ABB RAPID module: BE_User.sys

%%%
  VERSION:1
  LANGUAGE:ENGLISH
%%%

MODULE BE_User(SYSMODULE)
    !
    ! 2007-07-01 S?
    !   CHG: Added data for tcp check freq. from BE_Mnu.
    ! 2006-01-17 S?
    !   CHG: Added data scanMig and tdMig for use in setup.
    !   CHG: Renamed procedures due to name conflicts with bullseye.
    ! 2006-01-13 S?
    !   CHG: Changed name to BE_User due to restore problem with BullsEye, name conflict
    !
    TASK PERS tooldata tWeldGun:=[TRUE,[[0,0,0],[1,0,0,0]],[1,[1,0,0],[1,0,0,0],0,0,0]];
    !
    LOCAL CONST jointtarget jtEmpty:=[[9E+09,9E+09,9E+09,9E+09,9E+09,9E+09],[9E+09,9E+09,9E+09,9E+09,9E+09,9E+09]];
    TASK PERS jointtarget jtBEHome:=[[94.4267,-36.8911,24.1644,-0.0315949,63.4412,0.285663],[4816.37,9E+09,9E+09,9E+09,9E+09,9E+09]];
    TASK PERS jointtarget jtBEApprPos:=[[144.389,0.963088,5.42986,-3.28422,43.5331,5.14622],[4816.37,9E+09,9E+09,9E+09,9E+09,9E+09]];
    TASK PERS jointtarget jtBEStartPos:=[[143.497,1.4308,11.9387,-2.84858,36.5204,4.36587],[4816.37,9E+09,9E+09,9E+09,9E+09,9E+09]];
    !
    !CONST be_device devUp:=["sen1",TRUE,[6,45,100,100],[40,45,100,100],0.10,FALSE,TRUE,TRUE];
    CONST be_device devUp:=["sen1",TRUE,[6,45,100,100],[40,45,100,100],0.10,FALSE,TRUE,TRUE];
    CONST be_device devDown:=["sen1",TRUE,[6,45,100,100],[40,45,100,100],0.10,TRUE,TRUE,TRUE];
    CONST be_scan scanMig:=[2,8,8,45,35,25];
    !CONST be_tooldesign tdMig:=[TRUE,30,18,50,6,6,TRUE,TRUE,1.2,[150,120,100,100],[250,150,100,100]];
    CONST be_tooldesign tdMig:=[TRUE,30,18,40,6,6,TRUE,TRUE,1.2,[150,120,100,100],[250,150,100,100]];
    !
    TASK PERS num nTcpExtension:=20;
    ! vars for tcp check during production
    TASK PERS num nBECheckTcpFreq:=0;
    TASK PERS num nBECheckCycle:=0;
    TASK PERS num numElapsedTime:=607.948;
    TASK PERS num numMeanDev:=0.0669059;
    TASK PERS num numMaxDev:=0.0974435;

    !
    PROC BEToolSetup()
        VAR jointtarget jCurrPos;
        VAR string sHeader;
        VAR string sMsg{5};
        VAR btnres nAnswer;

        sHeader:="BullsEye"+" ("+GetTaskName()+")";
        MoveAbsJ [[94.4267,-36.8911,24.1644,-0.0315949,63.4412,0.285663],[4816.37,9E+09,9E+09,9E+09,9E+09,9E+09]]\NoEOffs, v1000, z50, toolWeldGun1;
        sMsg{1}:="Press Yes to run setup for BullsEye scanning process.";
        sMsg{2}:="";
        sMsg{3}:="Press No to cancel.";
        sMsg{4}:="";
        sMsg{5}:="";
        UIMsgBox\Header:=sHeader,sMsg{1}\MsgLine2:=sMsg{2}\MsgLine3:=sMsg{3}\MsgLine4:=sMsg{4}\MsgLine5:=sMsg{5}\Buttons:=btnYesNo\Icon:=iconInfo\Result:=nAnswer;
        IF (nAnswer=resYes) THEN
            !The length of the TCP extension, as measured from the end of the tool body, is defined
            !here in millimeters.
            sHeader:="BullsEye"+" ("+GetTaskName()+")";
            sMsg{1}:="TCP extension";
            sMsg{2}:="The length of the TCP extension, measured from the end of the tool body in mm.";
            sMsg{3}:="";
            sMsg{4}:="Current value: "+ValToStr(nTcpExtension);
            sMsg{5}:="Enter TCP extension (mm)";
            nTcpExtension:=UINumEntry(\Header:=sHeader\MsgArray:=sMsg\Icon:=iconInfo\InitValue:=nTcpExtension);

            sHeader:="BullsEye"+" ("+GetTaskName()+")";
            sMsg{1}:="Tool and positions";
            sMsg{2}:="";
            sMsg{3}:="Press Ok to modpos approach position, start position";
            sMsg{4}:="and select tool for BullsEye scanning process.";
            sMsg{5}:="";
            UIMsgBox\Header:=sHeader,sMsg{1}\MsgLine2:=sMsg{2}\MsgLine3:=sMsg{3}\MsgLine4:=sMsg{4}\MsgLine5:=sMsg{5}\Buttons:=btnOk\Icon:=iconInfo\Result:=nAnswer;

            Stop\NoRegain;
            ! modpos robtargets jtBEApprPos and jtBEStartPos
            MoveAbsJ jtBEHome\NoEOffs, v1000, z50, toolWeldGun1;
            ClkReset clockPartTimeConsume;
            ClkStart clockPartTimeConsume;
            BESetupToolJ jtBEApprPos,jtBEStartPos,nTcpExtension,tdMig,scanMig,devUp,v100,fine,toolWeldGun1\ElapsedTime:=numElapsedTime\MeanDev:=numMeanDev\MaxDev:=numMaxDev;
            Logging\INFO, "ElapsedTime="+ValToStr(numElapsedTime)+", MeanDev="+ValToStr(numMeanDev)+", MaxDev="+ValToStr(numMaxDev);
            toolWeldGun:=toolWeldGun1;
            toolLaser1.tload:=toolWeldGun1.tload;
            numTimeConsumeTotal:=ClkRead(clockPartTimeConsume);
            Logging\INFO, "BESetupToolJ: numTimeConsumeTotal="+ValToStr(numTimeConsumeTotal);
            ClkStop clockPartTimeConsume;
            MoveAbsJ jtBEHome\NoEOffs, v1000, z50, toolWeldGun1;
        ENDIF
    ENDPROC

    PROC BEToolCheck()
        ClkReset clockPartTimeConsume;
        ClkStart clockPartTimeConsume;
        BECheckTcp toolWeldGun1\XYZOnly\SingleScan;
        toolWeldGun:=toolWeldGun1;
        numTimeConsumeTotal:=ClkRead(clockPartTimeConsume);
        Logging\INFO, "BEToolCheck: numTimeConsumeTotal="+ValToStr(numTimeConsumeTotal);
        ClkStop clockPartTimeConsume;
    ENDPROC

    PROC BEToolUpdate()
        ClkReset clockPartTimeConsume;
        ClkStart clockPartTimeConsume;
        BEUpdateTcp toolWeldGun1\XYZOnly;
        toolWeldGun:=toolWeldGun1;
        numTimeConsumeTotal:=ClkRead(clockPartTimeConsume);
        Logging\INFO, "BEToolUpdate: numTimeConsumeTotal="+ValToStr(numTimeConsumeTotal);
        ClkStop clockPartTimeConsume;
    ENDPROC

    PROC BERefPnt()
        BERefPointer toolWeldGun1;
        toolWeldGun:=toolWeldGun1;
    ENDPROC

    PROC BEExtend()
        BETcpExtend toolWeldGun1\Absolute:=nTcpExtension;
        toolWeldGun:=toolWeldGun1;
    ENDPROC

ENDMODULE
